TYPE ST_RecipeBuilder_HMI :
    STRUCT
        Config  : ST_RecipeBuilder_Config;
		Limits  : ST_Recipe_Limits; 
    END_STRUCT
END_TYPE

(* stored: Version 1.1.0.1, ProductVersion 3.1.4024.15
   DUT ST_RecipeBuilder_HMI: Id {6eb6a18f-2a70-43f0-9365-d0b122d2f8c7} *)
